// TIA Portal V21 export
DATA_BLOCK "Pid_Sterilizzatore_RiscaldamentoAcqua"   // DB41
// stored: InstanceOfName PID_Compact, OfSystemLibElement PID_Compact, OfSystemLibVersion 2.4
PID_Compact   // technology object, version 2.4
   // VAR_INPUT
   //    Setpoint : Real := 20200.0;
   //    Input : Real := 20080.0;
   //    Input_PER : Int;
   //    Disturbance : Real;
   //    ManualEnable : Bool := FALSE;
   //    ManualValue : Real := 0.0;
   //    ErrorAck : Bool;
   //    Reset : Bool := FALSE;
   //    ModeActivate : Bool;
   // END_VAR
   // VAR_OUTPUT
   //    ScaledInput { ExternalWritable := 'False'} : Real := 20080.0;
   //    Output { ExternalWritable := 'False'} : Real := 3.174957;
   //    Output_PER { ExternalWritable := 'False'} : Int;
   //    Output_PWM { ExternalWritable := 'False'} : Bool := FALSE;
   //    SetpointLimit_H { ExternalWritable := 'False'} : Bool := FALSE;
   //    SetpointLimit_L { ExternalWritable := 'False'} : Bool := FALSE;
   //    InputWarning_H { ExternalWritable := 'False'} : Bool := FALSE;
   //    InputWarning_L { ExternalWritable := 'False'} : Bool := FALSE;
   //    State { ExternalWritable := 'False'} : Int := 3;
   //    Error { ExternalWritable := 'False'} : Bool;
   //    ErrorBits { ExternalWritable := 'False'} : DWord;
   // END_VAR
   // VAR_IN_OUT
   //    Mode : Int := 3;
   // END_VAR
   // VAR
   //    InternalDiagnostic : DWord;
   //    InternalVersion { ExternalWritable := 'False'} : DWord;
   //    InternalRTVersion : DWord;
   //    IntegralResetMode { S7_SetPoint := 'True'} : Int := 4;
   //    OverwriteInitialOutputValue : Real;
   //    RunModeByStartup { S7_SetPoint := 'True'} : Bool := TRUE;
   //    LoadBackUp : Bool;
   //    SetSubstituteOutput { S7_SetPoint := 'True'} : Bool := TRUE;
   //    PhysicalUnit { ExternalWritable := 'False'; S7_SetPoint := 'True'} : Int;
   //    PhysicalQuantity { ExternalWritable := 'False'; S7_SetPoint := 'True'} : Int := 1;
   //    ActivateRecoverMode { S7_SetPoint := 'True'} : Bool := TRUE;
   // END_VAR
   // VAR RETAIN
   //    Warning { ExternalWritable := 'False'} : DWord;
   //    WarningInternal { ExternalWritable := 'False'} : DWord;
   // END_VAR
   // VAR
   //    Progress { ExternalWritable := 'False'} : Real;
   //    CurrentSetpoint { ExternalWritable := 'False'} : Real;
   //    CancelTuningLevel { S7_SetPoint := 'True'} : Real := 10.0;
   //    SubstituteOutput { S7_SetPoint := 'True'} : Real := 1.5;
   //    Config { S7_SetPoint := 'True'} : PID_CompactConfig;
   //    CycleTime { S7_SetPoint := 'True'} : PID_CycleTime;
   //    CtrlParamsBackUp { S7_SetPoint := 'True'} : PID_CompactControlParams;
   //    PIDSelfTune { S7_SetPoint := 'True'} : PID_CompactSelfTune;
   //    PIDCtrl { S7_SetPoint := 'True'} : PID_CompactControl;
   // END_VAR
   // VAR RETAIN
   //    Retain { S7_SetPoint := 'True'} : PID_CompactRetain;
   // END_VAR
BEGIN
   Config.InputPerOn := FALSE;
   Config.InvertControl := FALSE;
   Config.InputUpperLimit := 100000.0;
   Config.InputLowerLimit := 0.0;
   Config.InputUpperWarning := 1000000.0;
   Config.InputLowerWarning := -100.0;
   Config.OutputUpperLimit := 9.0;
   Config.OutputLowerLimit := -5.0;
   Config.SetpointUpperLimit := 3.402822E+38;
   Config.SetpointLowerLimit := -3.402822E+38;
   Config.MinimumOnTime := 0.0;
   Config.MinimumOffTime := 0.0;
   Config.InputScaling.UpperPointIn := 27648.0;
   Config.InputScaling.LowerPointIn := 0.0;
   Config.InputScaling.UpperPointOut := 100.0;
   Config.InputScaling.LowerPointOut := 0.0;
   CycleTime.EnEstimation := TRUE;
   CycleTime.EnMonitoring := TRUE;
   CycleTime.Value := 0.009999501;
   CtrlParamsBackUp.Gain := 0.001;
   CtrlParamsBackUp.Ti := 0.15;
   CtrlParamsBackUp.Td := 0.0;
   CtrlParamsBackUp.TdFiltRatio := 0.1;
   CtrlParamsBackUp.PWeighting := 0.8;
   CtrlParamsBackUp.DWeighting := 0.0;
   CtrlParamsBackUp.Cycle := 0.02998491;
   PIDSelfTune.SUT.TuneRule := 0;
   PIDSelfTune.TIR.TuneRule := 0;
   Retain.CtrlParams.Gain := 0.004978305;
   Retain.CtrlParams.Ti := 1.655181;
   Retain.CtrlParams.Td := 0.4180084;
   Retain.CtrlParams.TdFiltRatio := 0.1;
   Retain.CtrlParams.PWeighting := 0.2609164;
   Retain.CtrlParams.DWeighting := 0.0;
   Retain.CtrlParams.Cycle := 0.0300108;
END_DATA_BLOCK
